VAR_GLOBAL CONSTANT
	/// "Index-Group/Offset", GET_SYMHANDLE_BYNAME
	cGET_SYMHANDLE_BYNAME: UDINT := 16#F003;
	/// "Index-Group/Offset", READ_WRITE_SYMVAL_BYHANDLE
	cREAD_WRITE_SYMVAL_BYHANDLE: UDINT := 16#F005;
END_VAR

(* stored: Version 1.1.0.1, ProductVersion 3.1.0.19
   GVL ADS_IndexGroup: Id {0bd41315-2e3d-4828-93ba-156c7efe43b2} *)
